PROGRAM Firebird_ReadAlarms
VAR_INPUT
	ParamTimeBetweenReconnect	: TIME := T#1M;
	IN_StartRead				: BOOL;
	IN_FrequencyRead			: TIME := T#1M;
	IN_bAct						: BOOL; // Read only Active values
	IN_FilterAct				: BOOL;
	IN_bAck						: BOOL; // Read only Acknowledged values
	IN_FilterAck				: BOOL;
	
	IN_TimeStampStart			: TIMESTRUCT;
	IN_TimeStampEnd				: TIMESTRUCT;
	
END_VAR
VAR CONSTANT
	NbMaxElements	 			: UINT := 250;
END_VAR
VAR_OUTPUT
	OUT_Busy					: BOOL;
	
END_VAR
VAR
	
	AX_Buffer_Alarms			: ARRAY[1..NbMaxElements] OF St_AlarmsV2;		// Buffer of alarms to write
	StNull						: St_AlarmsV2;		// Buffer of alarms to write
		
	// Connexion
		TP_Reconnect			: TP;
		Trig_Connect			: R_TRIG;
		TRIG_CmdStart			: R_TRIG;
		RS_Connect				: RS;
		RS_HasBeenConnected		: RS;
	// DISCONNECT
		TrigStartDisconnect				: R_TRIG;
		RsStartDisconnect				: RS;		
			
	// READ File       
		TP_ReadBddPeriodically	: TP;
		TRIG_ReadBddPeriodically: R_TRIG;

		ETAPE					: UINT;
		Trig_Start				: R_TRIG;   
		RS_Start				: RS; 	
		Requete					: ARRAY[1..10] OF STRING(1000);
		RequeteNull				: ARRAY[1..10] OF STRING(1000);
		sToAdd					: STRING(1000);
		pPosRequete				: DINT;
		TimeStampNull			: TIMESTRUCT;
		TimeStampDefault		: TIMESTRUCT;
		sTimeStampStart			: STRING(255);
		sTimeStampEnd			: STRING(255);
		sValue					: STRING(255);
		sAck					: STRING(255);
		Format					: FB_FormatString;
		SQLDatabase				: FB_SQLDatabaseEvt('',T#10S);
		SQLCommand				: FB_SQLCommandEvt('',T#10S);
		SQLCommandNull			: FB_SQLCommandEvt('',T#10S);
		SQLResult				: FB_SQLResultEvt('',T#10S);
		
	
	// General variables
		nbMax					: UINT;
		bInit 					: BOOL;
		NomTableAlarms			: STRING(255) := 'TABLE_ALARMS_V2';
		KK						: UINT;
		
	//TABLEAU
	
		AX_MesAlarmCode_Bool	: ARRAY [1..CstNbAlarmCode] OF ARRAY[1..15] OF BOOL; //Tableau de tous les alarmesCode en Bool
		AX_Alarm_State			: ARRAY [1..CstNbAlarmCode] OF ARRAY[1..15] OF BOOL; //Tableau de Bool avec toutes les nouveaux bit modifiés
		AX_MesAck				: ARRAY [1..CstNbAlarmCode] OF ARRAY[1..15] OF BOOL;
		AX_Ack_State			: ARRAY [1..CstNbAlarmCode] OF ARRAY[1..15] OF BOOL; //Tableau de Bool avec tous les nouveaux acknowledgement 

	

END_VAR

// DataProcessing
IF NOT bInit THEN
	M_Init();
END_IF
RS_HasBeenConnected(SET := SQLDatabase.bConnected);
TP_Reconnect(In :=RS_HasBeenConnected.Q1 AND NOT SQLDatabase.bConnected OR NOT bInit OR TP_Reconnect.Q, PT := ParamTimeBetweenReconnect);
	
TP_ReadBddPeriodically(IN := NOT TP_ReadBddPeriodically.Q, PT := IN_FrequencyRead);
TRIG_ReadBddPeriodically(CLK := TP_ReadBddPeriodically.Q);
TRIG_CmdStart(CLK := IN_StartRead);

Trig_Start(CLK := SQLDatabase.bConnected AND NOT OUT_Busy AND ( TRIG_CmdStart.Q OR TRIG_ReadBddPeriodically.Q));
IF Trig_Start.Q THEN
	// Init the table :
	FOR KK := 1 TO 10 DO 
		Requete[KK] := RequeteNull[KK];
	END_FOR
	FOR KK := 1 TO NbMaxElements DO
		AX_Buffer_Alarms[KK] := StNull;
	END_FOR
	Requete := RequeteNull;
	nbMax := NbMaxElements;
	pPosRequete := 0;
	// Je commence par préparer ma requête 
	IF MEMCMP(pBuf1 := ADR(IN_TimeStampStart), pBuf2:=ADR(TimeStampNull), n:=SIZEOF(TimeStampNull))=0 THEN
		IN_TimeStampStart := TimeStampDefault;
	END_IF
	sTimeStampStart := systemtime_to_string(in := IN_TimeStampStart);
	sTimeStampEnd := systemtime_to_string(in := IN_TimeStampEnd);
	Format( sFormat := 'Select first %d "TIMESTAMP_START", case when "TIMESTAMP_STOP" is null then cast($'01.01.1970, 00:00:00.000$' as timestamp) else "TIMESTAMP_STOP" end,AlarmsID,Act,Ack from %s where "TIMESTAMP_START" > $'%s$' ', 
		sOut=> sToAdd,
		arg1 := F_UINT(In:=nbMax),
		arg2 := F_STRING(In := NomTableAlarms),
		arg3 := F_STRING(in := sTimeStampStart)
	);
	MEMCPY(destAddr := ADR(requete), srcAddr := ADR(sToAdd), n := SIZEOF(sToAdd));
	pPosRequete:= pPosRequete + LEN(STR := sToAdd);
	
	IF IN_FilterAct THEN
		sToAdd := CONCAT(STR1 := ' AND Act = ', STR2 := UINT_TO_STRING(BOOL_TO_UINT(IN_bAct)));
		MEMCPY(srcAddr:= ADR(sToAdd), destAddr := ADR(Requete)+DINT_TO_DWORD(pPosRequete), n:= SIZEOF(sToAdd));
		pPosRequete:= pPosRequete + LEN(STR := sToAdd);
	END_IF
	
	IF IN_FilterAck THEN
		sToAdd := CONCAT(STR1 := ' AND Ack = ', STR2 := UINT_TO_STRING(BOOL_TO_UINT(IN_bAck)));
		MEMCPY(srcAddr:= ADR(sToAdd), destAddr := ADR(Requete)+DINT_TO_DWORD(pPosRequete), n:= SIZEOF(sToAdd));
		pPosRequete:= pPosRequete + LEN(STR := sToAdd);
	END_IF	

	sToAdd := ' order by TIMESTAMP_START desc';
	MEMCPY(srcAddr:= ADR(sToAdd), destAddr := ADR(Requete)+DINT_TO_DWORD(pPosRequete), n:= SIZEOF(sToAdd));
	pPosRequete:= pPosRequete + LEN(STR := sToAdd);	
	ETAPE := 1;
END_IF
		
CASE ETAPE OF
	1: // CONNECTED
		OUT_Busy := TRUE;
		IF SQLDatabase.CreateCmd(pSQLCommand := ADR(SQLCommand)) THEN 
			IF NOT SQLCommAND bError THEN
				ETAPE := 2;
			ELSIF SQLCommAND bError THEN
				ETAPE := 255;
			END_IF
		END_IF
		
	2:	
		IF SQLCommAND ExecuteDataReturn(pSQLCmd := ADR(Requete), cbSQLCmd := SIZEOF(Requete), pSQLDBResult := ADR(SQLResult))THEN
			IF  NOT SQLCommAND bError THEN
				ETAPE := 3;
			ELSIF SQLCommAND bError THEN
				ETAPE := 255;
			END_IF
		END_IF
	3: 
		IF SQLResult.Read(nStartIndex := 1, nRecordCount := NbMaxElements, pData := ADR(AX_Buffer_Alarms), cbData := SIZEOF(AX_Buffer_Alarms), bDataRelease := TRUE, bWithVerifying := FALSE) THEN
			IF NOT SQLResult.bError THEN
				Etape := 4;
			ELSE
				ETAPE := 255;
			END_IF
		END_IF
	4:
		IF NOT SQLDatabase.bError THEN

			Requete  := RequeteNull;
			Trig_Start(CLK := FALSE);
			Etape := 0;
			OUT_Busy := FALSE;
		ELSE 
			ETAPE := 255;
		END_IF
	255: 
		OUT_Busy := FALSE;
		Requete := RequeteNull;
		Etape := 0;
		IN_StartRead := FALSE;
END_CASE

METHOD M_Connect : BOOL

VAR_OUTPUT
END_VAR
VAR_INPUT
	IN_hDBID				: DINT;
	IN_Start				: BOOL;
END_VAR
Trig_Connect(CLK := IN_Start);
RS_Connect(SET := Trig_Connect.Q);
IF RS_Connect.Q1 THEN
	IF SQLDatabase.Connect(hDBID := IN_hDBID) THEN;
		RS_Connect(RESET1 := TRUE);
		RS_Connect(RESET1 := FALSE);
	END_IF
END_IF
END_METHOD

METHOD M_Disconnect : BOOL
VAR_INPUT
END_VAR
VAR_INPUT
	IN_Start				: BOOL;
END_VAR
TrigStartDisconnect(CLK := IN_Start);
RsStartDisconnect(SET := TrigStartDisconnect.Q);
IF RsStartDisconnect.Q1 THEN
	IF SQLDatabase.Disconnect() THEN;
		RsStartDisconnect(RESET1 := TRUE);
		RsStartDisconnect(RESET1 := FALSE);
	END_IF
END_IF
END_METHOD

METHOD M_Init

VAR
	LL	: SINT;
	KK 	: SINT;
END_VAR
TimeStampDefault.wYear := 1995;
TimeStampDefault.wMonth := 3;
TimeStampDefault.wDay := 12;

bInit := TRUE;
END_METHOD

END_PROGRAM

(* stored: Version 1.1.0.1, ProductVersion 3.1.4024.6
   POU Firebird_ReadAlarms: Id {93dbf52d-bd1f-4f0f-be28-6d084e03bfe0}, SpecialFunc None
   Method M_Connect: Id {3f144ec5-1b4b-4d23-8d57-af6b4c9ff6ad}
   Method M_Disconnect: Id {113491eb-e2fc-4277-803b-42a5777d26f7}
   Method M_Init: Id {ce7c8b10-4ea8-4bb2-93fd-1b4cb5340497} *)
